// TIA Portal V18 export
DATA_BLOCK "SS1_A6_16DI_DI_Vars"   // DB11061
{ S7_Optimized_Access := 'FALSE' }
VERSION : 0.1
// stored: AutoNumber false, DBAccessibleFromOPCUA true, IsOnlyStoredInLoadMemory false, IsWriteProtectedInAS false
   VAR
      DI1 : "UDT_DIadv";
      DI2 : "UDT_DIadv";
      DI3 : "UDT_DIadv";
      DI4 : "UDT_DIadv";
      DI5 : "UDT_DIadv";
      DI6 : "UDT_DIadv";
      DI7 : "UDT_DIadv";
      DI8 : "UDT_DIadv";
      DI9 { S7_SetPoint := 'True'} : "UDT_DIadv";
      DI10 { S7_SetPoint := 'True'} : "UDT_DIadv";
      DI11 { S7_SetPoint := 'True'} : "UDT_DIadv";
      DI12 { S7_SetPoint := 'True'} : "UDT_DIadv";
      DI13 { S7_SetPoint := 'True'} : "UDT_DIadv";
      DI14 { S7_SetPoint := 'True'} : "UDT_DIadv";
      DI15 { S7_SetPoint := 'True'} : "UDT_DIadv";
      DI16 { S7_SetPoint := 'True'} : "UDT_DIadv";
   END_VAR
BEGIN
   DI1.cFuncSystemID := 100;
   DI1.cFuncVar := 1;
   DI2.cFuncSystemID := 100;
   DI2.cFuncVar := 3;
   DI5.cFuncSystemID := 100;
   DI5.cFuncVar := 5;
   DI6.cFuncSystemID := 100;
   DI6.cFuncVar := 6;
END_DATA_BLOCK
